PROGRAM P03_MachineControl
VAR
	tonStarting					:TON;
	tonStopping					:TON;
	tonRobotStarting			:TON;
	tonRobotStopping			:TON;
	tonRobotInitialising		:TON;
	
	bStop						:BOOL;
	
	fbBatch						:FB_Batch;
	tonBatchTime				:FB_TONP;
END_VAR
VAR // added by the converter: edge detectors and wires of the graphical bodies
    _w1, _w2, _w3, _w4, _w5, _w6, _w7, _w8, _w9, _w10, _w11, _w12 : BOOL;
    _rt1 : R_TRIG;
END_VAR

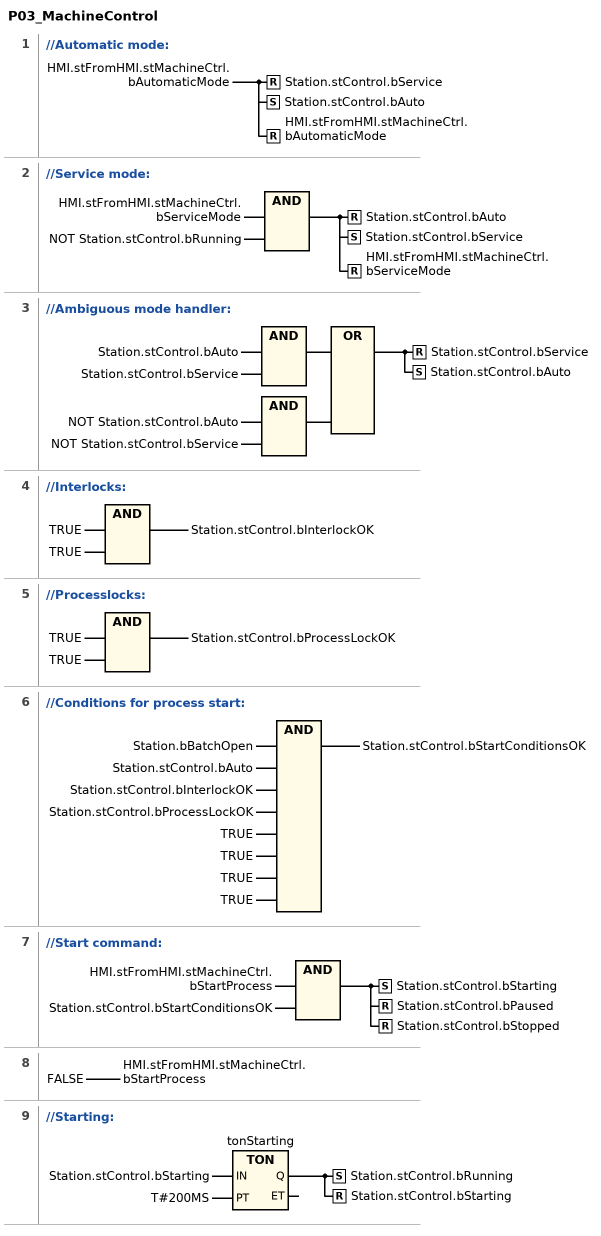
// NETWORK 1
// label: //Automatic mode
Station.stControl.bService R= HMI.stFromHMI.stMachineCtrl.bAutomaticMode;
Station.stControl.bAuto S= HMI.stFromHMI.stMachineCtrl.bAutomaticMode;
HMI.stFromHMI.stMachineCtrl.bAutomaticMode R= HMI.stFromHMI.stMachineCtrl.bAutomaticMode;

// NETWORK 2
// label: //Service mode
_w1 := HMI.stFromHMI.stMachineCtrl.bServiceMode AND (NOT Station.stControl.bRunning);
Station.stControl.bAuto R= _w1;
Station.stControl.bService S= _w1;
HMI.stFromHMI.stMachineCtrl.bServiceMode R= _w1;

// NETWORK 3
// label: //Ambiguous mode handler
_w2 := Station.stControl.bAuto AND Station.stControl.bService OR (NOT Station.stControl.bAuto) AND (NOT Station.stControl.bService);
Station.stControl.bService R= _w2;
Station.stControl.bAuto S= _w2;

// NETWORK 4
// label: //Interlocks
Station.stControl.bInterlockOK := TRUE AND TRUE;

// NETWORK 5
// label: //Processlocks
Station.stControl.bProcessLockOK := TRUE AND TRUE;

// NETWORK 6
// label: //Conditions for process start
Station.stControl.bStartConditionsOK := Station.bBatchOpen AND Station.stControl.bAuto AND Station.stControl.bInterlockOK AND Station.stControl.bProcessLockOK AND TRUE AND TRUE AND TRUE AND TRUE;

// NETWORK 7
// label: //Start command
_w3 := HMI.stFromHMI.stMachineCtrl.bStartProcess AND Station.stControl.bStartConditionsOK;
Station.stControl.bStarting S= _w3;
Station.stControl.bPaused R= _w3;
Station.stControl.bStopped R= _w3;

// NETWORK 8
HMI.stFromHMI.stMachineCtrl.bStartProcess := FALSE;

// NETWORK 9
// label: //Starting
tonStarting(IN := Station.stControl.bStarting, PT := T#200MS); // TON
Station.stControl.bRunning S= tonStarting.Q;
Station.stControl.bStarting R= tonStarting.Q;

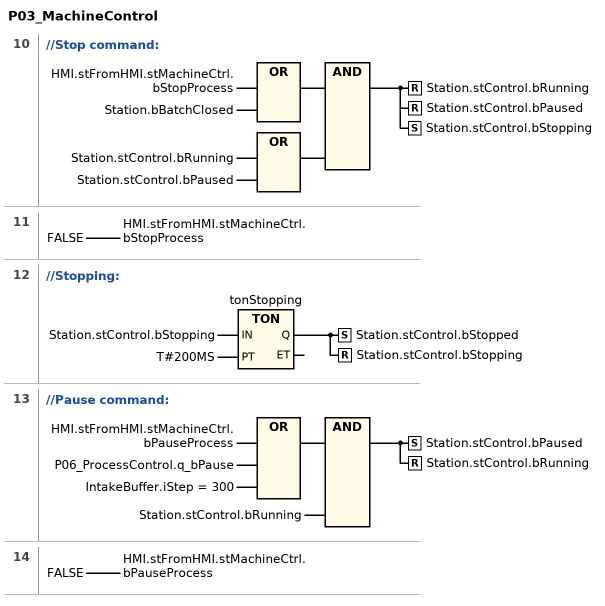
// NETWORK 10
// label: //Stop command
_w4 := (HMI.stFromHMI.stMachineCtrl.bStopProcess OR Station.bBatchClosed) AND (Station.stControl.bRunning OR Station.stControl.bPaused);
Station.stControl.bRunning R= _w4;
Station.stControl.bPaused R= _w4;
Station.stControl.bStopping S= _w4;

// NETWORK 11
HMI.stFromHMI.stMachineCtrl.bStopProcess := FALSE;

// NETWORK 12
// label: //Stopping
tonStopping(IN := Station.stControl.bStopping, PT := T#200MS); // TON
Station.stControl.bStopped S= tonStopping.Q;
Station.stControl.bStopping R= tonStopping.Q;

// NETWORK 13
// label: //Pause command
_w5 := (HMI.stFromHMI.stMachineCtrl.bPauseProcess OR P06_ProcessControl.q_bPause OR (IntakeBuffer.iStep = 300)) AND Station.stControl.bRunning;
Station.stControl.bPaused S= _w5;
Station.stControl.bRunning R= _w5;

// NETWORK 14
HMI.stFromHMI.stMachineCtrl.bPauseProcess := FALSE;

ACTION Batch:
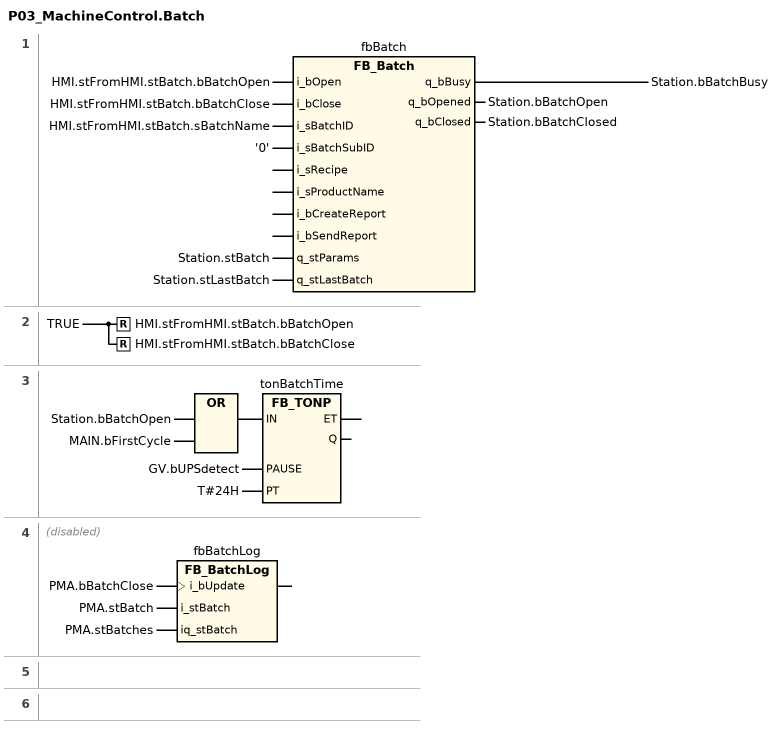
// NETWORK 1
fbBatch(
    i_bOpen := HMI.stFromHMI.stBatch.bBatchOpen,
    i_bClose := HMI.stFromHMI.stBatch.bBatchClose,
    i_sBatchID := HMI.stFromHMI.stBatch.sBatchName,
    i_sBatchSubID := '0',
    q_stParams := Station.stBatch,
    q_stLastBatch := Station.stLastBatch,
    q_bOpened => Station.bBatchOpen,
    q_bClosed => Station.bBatchClosed); // FB_Batch
Station.bBatchBusy := fbBatch.q_bBusy;

// NETWORK 2
HMI.stFromHMI.stBatch.bBatchOpen R= TRUE;
HMI.stFromHMI.stBatch.bBatchClose R= TRUE;

// NETWORK 3
tonBatchTime(IN := Station.bBatchOpen OR MAIN.bFirstCycle, PAUSE := GV.bUPSdetect, PT := T#24H); // FB_TONP

// NETWORK 4 (disabled)
// _rt1(CLK := PMA.bBatchClose);
// fbBatchLog(i_bUpdate := _rt1.Q, i_stBatch := PMA.stBatch, iq_stBatch := PMA.stBatches); // FB_BatchLog

// NETWORK 5

// NETWORK 6
END_ACTION

ACTION Robot:
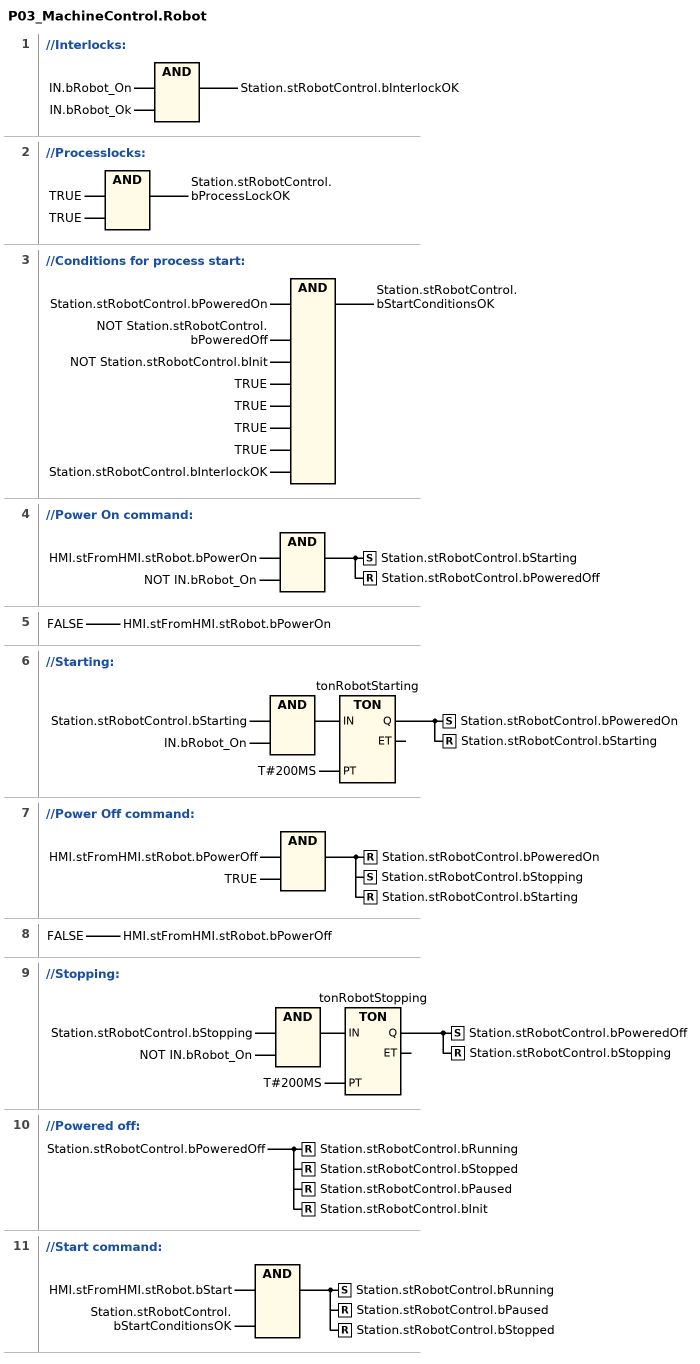
// NETWORK 1
// label: //Interlocks
Station.stRobotControl.bInterlockOK := IN.bRobot_On AND IN.bRobot_Ok;

// NETWORK 2
// label: //Processlocks
Station.stRobotControl.bProcessLockOK := TRUE AND TRUE;

// NETWORK 3
// label: //Conditions for process start
Station.stRobotControl.bStartConditionsOK := Station.stRobotControl.bPoweredOn AND (NOT Station.stRobotControl.bPoweredOff) AND (NOT Station.stRobotControl.bInit) AND TRUE AND TRUE AND TRUE AND TRUE AND Station.stRobotControl.bInterlockOK;

// NETWORK 4
// label: //Power On command
_w6 := HMI.stFromHMI.stRobot.bPowerOn AND (NOT IN.bRobot_On);
Station.stRobotControl.bStarting S= _w6;
Station.stRobotControl.bPoweredOff R= _w6;

// NETWORK 5
HMI.stFromHMI.stRobot.bPowerOn := FALSE;

// NETWORK 6
// label: //Starting
tonRobotStarting(IN := Station.stRobotControl.bStarting AND IN.bRobot_On, PT := T#200MS); // TON
Station.stRobotControl.bPoweredOn S= tonRobotStarting.Q;
Station.stRobotControl.bStarting R= tonRobotStarting.Q;

// NETWORK 7
// label: //Power Off command
_w7 := HMI.stFromHMI.stRobot.bPowerOff AND TRUE;
Station.stRobotControl.bPoweredOn R= _w7;
Station.stRobotControl.bStopping S= _w7;
Station.stRobotControl.bStarting R= _w7;

// NETWORK 8
HMI.stFromHMI.stRobot.bPowerOff := FALSE;

// NETWORK 9
// label: //Stopping
tonRobotStopping(IN := Station.stRobotControl.bStopping AND (NOT IN.bRobot_On), PT := T#200MS); // TON
Station.stRobotControl.bPoweredOff S= tonRobotStopping.Q;
Station.stRobotControl.bStopping R= tonRobotStopping.Q;

// NETWORK 10
// label: //Powered off
_w8 := Station.stRobotControl.bPoweredOff;
Station.stRobotControl.bRunning R= _w8;
Station.stRobotControl.bStopped R= _w8;
Station.stRobotControl.bPaused R= _w8;
Station.stRobotControl.bInit R= _w8;

// NETWORK 11
// label: //Start command
_w9 := HMI.stFromHMI.stRobot.bStart AND Station.stRobotControl.bStartConditionsOK;
Station.stRobotControl.bRunning S= _w9;
Station.stRobotControl.bPaused R= _w9;
Station.stRobotControl.bStopped R= _w9;

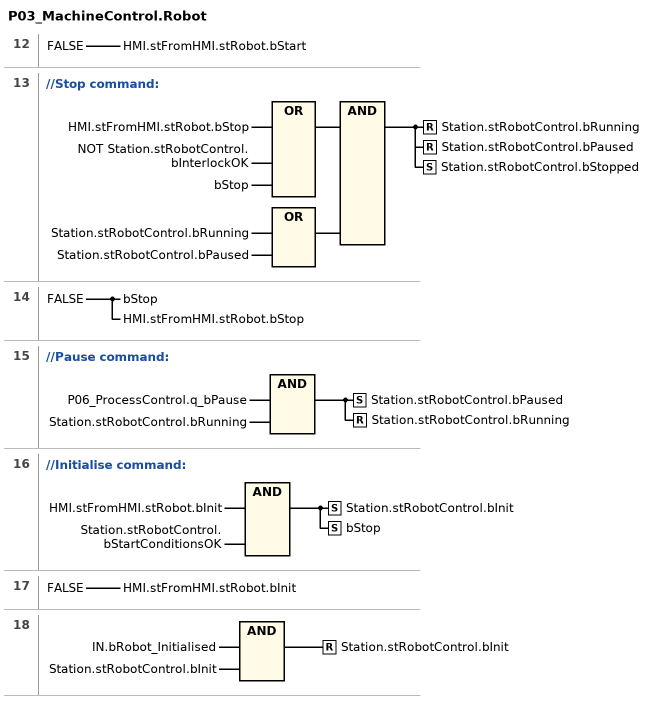
// NETWORK 12
HMI.stFromHMI.stRobot.bStart := FALSE;

// NETWORK 13
// label: //Stop command
_w10 := (HMI.stFromHMI.stRobot.bStop OR (NOT Station.stRobotControl.bInterlockOK) OR bStop) AND (Station.stRobotControl.bRunning OR Station.stRobotControl.bPaused);
Station.stRobotControl.bRunning R= _w10;
Station.stRobotControl.bPaused R= _w10;
Station.stRobotControl.bStopped S= _w10;

// NETWORK 14
bStop := FALSE;
HMI.stFromHMI.stRobot.bStop := FALSE;

// NETWORK 15
// label: //Pause command
_w11 := P06_ProcessControl.q_bPause AND Station.stRobotControl.bRunning;
Station.stRobotControl.bPaused S= _w11;
Station.stRobotControl.bRunning R= _w11;

// NETWORK 16
// label: //Initialise command
_w12 := HMI.stFromHMI.stRobot.bInit AND Station.stRobotControl.bStartConditionsOK;
Station.stRobotControl.bInit S= _w12;
bStop S= _w12;

// NETWORK 17
HMI.stFromHMI.stRobot.bInit := FALSE;

// NETWORK 18
Station.stRobotControl.bInit R= IN.bRobot_Initialised AND Station.stRobotControl.bInit;
END_ACTION

END_PROGRAM

(* stored: Version 1.1.0.1
   POU P03_MachineControl: Id {87ffe191-cc71-433a-bb1a-f71bbc002b19}, SpecialFunc None
   Action Batch: Id {79893817-f028-4f62-9cea-6c40e9a77ed5}
   Action Robot: Id {5bff24de-b9d1-4649-add2-25a211008589} *)
